GLOBALCONSTANTS IG2_Source_Addresses (* Industry Group 2 specific source addresses *)
  (* Standard: 61499-1 *)
  (* Version 1.0, 2026-06-29, Franz Höpfinger, Demmler Andreas Fahrzeugbau *)
  PACKAGE isobus::pgn::const;
  VAR_GLOBAL CONSTANT
    SA_RESERVED_128 : BYTE := 128; (* Source Address: thru 235 are reserved by ISO for the self-configurable address capability - All *)
    SA_DATA_LOGGER : BYTE := 236; (* Source Address: Data Logger - A data logging server that provides the LOG functionality as *)
    SA_TIM_SERVER : BYTE := 237; (* Source Address: TIM Server - Control function that represents a Tractor Implement Management *)
    SA_SEQUENCE_CONTROLLER : BYTE := 238; (* Source Address: Sequence Controller - The master in the Sequence Control System as defined in *)
    SA_POSITION_CONTROL : BYTE := 239; (* Source Address: Position Control - Multiple axis position control of a devices movable device *)
    SA_TRACTOR_ECU : BYTE := 240; (* Source Address: Tractor ECU - A gateway (see ISO 11783-4) between the tractor and the implement *)
    SA_TAILINGS_MONITORING : BYTE := 241; (* Source Address: Tailings Monitoring - Monitoring of the quantity of unthreshed material returned *)
    SA_HEADER_CONTROL : BYTE := 242; (* Source Address: Header Control - Control of the headers reel rate and material delivery rate *)
    SA_PRODUCT_LOSS_MONITORING : BYTE := 243; (* Source Address: Product Loss Monitoring - Monitoring of the amount of produce being lost from *)
    SA_PRODUCT_MOISTURE_SENSING : BYTE := 244; (* Source Address: Product Moisture Sensing - Monitoring of the produce moisture content *)
    SA_NON_VIRTUAL_TERMINAL_DISPLAY_IMPLEMENT_BUS : BYTE := 245; (* Source Address: Non Virtual Terminal Display (Implement Bus) - A non Virtual Terminal cab display *)
    SA_OPERATOR_CONTROLS_MACHINE_SPECIFIC : BYTE := 246; (* Source Address: Operator Controls - Machine Specific - Non auxiliary operator control inputs *)
    SA_TASK_CONTROL_MAPPING_COMPUTER : BYTE := 247; (* Source Address: Task Control (Mapping Computer) - A control function on the 11783 network that is *)
  END_VAR
END_GLOBALCONSTANTS
